FUNCTION nota_hiz_donusturucu : REAL
VAR_INPUT
	nota :REAL;
	offset : REAL;
END_VAR

nota_hiz_donusturucu := LIMIT(0, (((((nota + offset)+8.845)*((nota + offset)+8.845)/9.708) + 29.03139) * 100), 8800);

END_FUNCTION

(* stored: Version 1.1.0.1
   POU nota_hiz_donusturucu: Id {aed1288b-1585-4b47-8ee7-f8035076d6a2}, SpecialFunc None *)
